ADAPTER Adapter (* Adapter Interface *)
  (* Standard: 61499-1 *)
  (* Version 0.0, 2008-04-22, GE, 4DIAC-Consortium *)
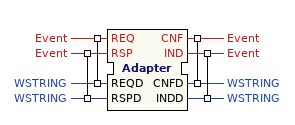
  EVENT_INPUT
    REQ WITH REQD; (* Request from Socket *)
    RSP WITH RSPD; (* Response from Socket *)
  END_EVENT
  EVENT_OUTPUT
    CNF WITH CNFD; (* Confirmation from Plug *)
    IND WITH INDD; (* Indication from Plug *)
  END_EVENT
  VAR_INPUT
    REQD : WSTRING; (* Request Data from Socket *)
    RSPD : WSTRING; (* Response Data from Socket *)
  END_VAR
  VAR_OUTPUT
    CNFD : WSTRING; (* Confirmation Data from Plug *)
    INDD : WSTRING; (* Indication Data from Plug *)
  END_VAR
  SERVICE PLUG/SOCKET
    SEQUENCE request_confirm
      SOCKET.REQ(REQD) -> PLUG.REQ(REQD);
      PLUG.CNF(CNFD) -> SOCKET.CNF(CNFD);
    END_SEQUENCE
    SEQUENCE indication_response
      PLUG.IND(INDD) -> SOCKET.IND(INDD);
      SOCKET.RSP(RSPD) -> PLUG.RSP(RSPD);
    END_SEQUENCE
  END_SERVICE
END_ADAPTER
